(* CODESYS project e!C_Alarm_Test_1.ecp

Project tree, tasks and I/O mapping:
  Controller : 750-8202 PFC200 2ETH RS, WAGO, order no. 0750-8202, version 5.11.1.16
    application Application
      libraries: Util, * (System)
      task PLC_Task (cyclic, interval t#10ms, priority 14) calls PLC_PRG
      task AlarmManagerTask (cyclic, interval 50 ms, priority 15) calls AlarmManager.Alarm_Prg
      task VISU_TASK (cyclic, interval 100 ms, priority 15) calls VisuElems.Visu_Prg
      program PLC_PRG [ST]
      Alarm_Configuration
        alarm class Error (priority 10, acknowledge REP_ACK)
        alarm class Warning (priority 30, acknowledge REP)
        alarm class Info (priority 100, acknowledge REP)
        AlarmStorage
        text list AlarmGroup
        alarm group AlarmGroup
            0 [Error]: Comparison Equal, ExpressionToCompare TRUE, Expression PLC_PRG.xAlarmEvent1 - "Alarm Text 1..."
      visualisation Visualization
    DeviceAdapter
    Kbus : Kbus, WAGO, version 1.4.0.2
        unmapped channels: K-BUS diagnostics
    MODBUS
      MODBUS : MODBUS, WAGO, order no. n/a, version 1.1.1.15
    Serial
      COM1 : COM1, WAGO, version 0.0.0.19
  libraries: VisuSymbols, 3.5.10.0 (System); WagoVisuIcons, 1.0.0.8 (WAGO)
  text list GlobalTextList
*)

// Controller/Application/PLC_PRG
PROGRAM PLC_PRG
VAR
	AlarmTrigger1: BLINK;
	xAlarmEvent1: BOOL;
	xAlarmEnable: BOOL := TRUE;
	tAlarmLow: TIME := T#2s;
	tAlarmHigh: TIME := T#2s;
END_VAR



AlarmTrigger1(ENABLE:= xAlarmEnable, TIMELOW:= tAlarmLow, TIMEHIGH:= tAlarmHigh, OUT=> xAlarmEvent1);

END_PROGRAM

// Controller/Application/Visualization
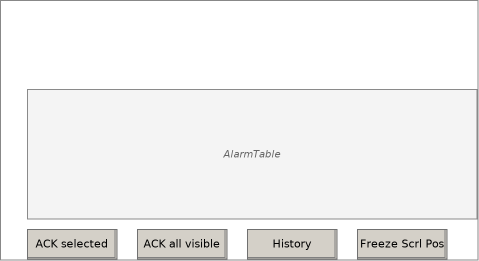
VISUALIZATION Visualization  // 479x261
VAR_IN_OUT
END_VAR
VAR
	bAckSel : BOOL;
	bAckVisible : BOOL;
	bHistory : BOOL;
	bFreezeScrlPos : BOOL;
END_VAR
    AlarmTable (27,89 450x130)
        Column[0]: ColumnTitle=Timestamp
        Column[1]: ColumnTitle=Message
        p1521930926: AlarmGroup
        p1663851261: Error
        p428520879: bAckSel
        p2607059081: bAckVisible
        p3266827225: bHistory
        p3894972949: bFreezeScrlPos
    Button (27,229 90x30), "ACK selected"
        toggle bAckSel
    Button (137,229 90x30), "ACK all visible"
        toggle bAckVisible
    Button (247,229 90x30), "History"
        toggle bHistory
    Button (357,229 90x30), "Freeze Scrl Pos"
        toggle bFreezeScrlPos
END_VISUALIZATION

(* text list AlarmGroup (id | default)
  0 | Alarm Text 1...
   |  *)
